{attribute 'GeneratedUsingTerminal: EP7211-0034-0029'}
{attribute addProperty BoxType "EP7211-0034-0029"}
{attribute addProperty Id "AdsAddrAT %I*.TcoAmsAddr0DcOutputShiftAT %I*DINT4DcInputShiftAT %I*DINT4Chn0AT %I*USINT1StateAT %I*UINT2"}
{attribute addProperty CRC "3737110711"}
{attribute addProperty Size "11"}
TYPE InfoData_DEBFC8B7 :
STRUCT
	{attribute addProperty Name "AdsAddr"}
	AdsAddr AT %I* : .TcoAmsAddr;
	{attribute addProperty Name "DcOutputShift"}
	DcOutputShift AT %I* : DINT;
	{attribute addProperty Name "DcInputShift"}
	DcInputShift AT %I* : DINT;
	{attribute addProperty Name "Chn0"}
	Chn0 AT %I* : USINT;
	{attribute addProperty Name "State"}
	State AT %I* : UINT;
END_STRUCT
END_TYPE

(* stored: Version 1.2.0.0, ProductVersion 3.1.4024.9
   DUT InfoData_DEBFC8B7: Id {e56098a6-ebeb-41ce-8946-7fc9f792e81c} *)
